INTERFACE I_DatatypePack

METHOD PUBLIC Register
VAR_INPUT
	Marshallers : I_GraphDatatypes;
END_VAR
END_METHOD

END_INTERFACE

(* stored: Version 1.1.0.1, ProductVersion 3.1.4024.12
   Itf I_DatatypePack: Id {c60741ea-3237-0ac6-2f76-f10f1e446198}
   Method Register: Id {a50b900d-258c-08bb-3c09-dc93df12a0ea} *)
